Universal Robots PolyScope program: browser.urp

Program browser (installation=cube_dev1 directory=/programs/cube createdIn=5.11.5.1010327 lastSavedIn=5.11.5.1010327 robotSerialNumber=20215500677)
Calibrated DH parameters: a=[0.000204, -0.239222, -0.391845, -0.000001, 0.000022, 0]; d=[0.162722, -355.808559, 353.37206, 2.570385, 0.099741, 0.099629]; alpha=[1.571124, 0.000988, 0.008295, 1.568963, -1.570303, 0]; deltaTheta=[0, -0.973091, 7.204745, 0.05153, 0, 0]
BeforeStart
  MoveJ speed 120 deg/s, acceleration 120 deg/s^2 (useActiveTCP=false) tcp=SandTCP; feature=Point_1
    Waypoint Sand_Base: TCP in base x=-341.949 y=196.192 z=697.874 mm, rx=0 ry=0 rz=-1.5708 rad; joints [-57.163, -82.73, 107.731, 93.373, -53.983, -132.185] deg; TCP offset x=1.003 y=125.541 z=104.154 mm, rx=-0.7854 ry=0 rz=0 rad; feature pose in base x=-341.965 y=196.202 z=697.85 mm, rx=0 ry=0 rz=-1.5843 rad
Robot Program (runOnlyOnce=false)
  Wait Sleep waitTime=0.01
Event  expression=PinsBtn≟ True
  Folder Sand
    MoveL speed 50 mm/s, acceleration 1200 mm/s^2 (useActiveTCP=false) tcp=SandTCP; feature=Base
      MoveDirectionNode (selectedDirection=ZPlus)
        Until TOOL_CONTACT_DETECTION (allowActions=false retraction=0.001 decelerationAcceleration=3 decelerationAngularAcceleration=34.906585)
      URCap Finishing Tool Control (Robotiq_Copilot, Robotiq Inc.) dataModel(ToolOutputNameKey=SanderOn, HackTriggeringContributionIsDefinedMethodKey=true)
    MoveL speed 50 mm/s, acceleration 1200 mm/s^2 (useActiveTCP=true) feature=Base
      Force Simple feature=Base; selection=[0, 0, 1, 0, 0, 0]; wrench=[0, 0, 5, 0, 0, 0]; limitsForce=[0.15, 0.15, 0.15, 1.047198, 1.047198, 1.047198]; limitsMotion=[0.1, 0.1, 0.1, 0.349066, 0.349066, 0.349066]
        MoveDirectionNode (selectedDirection=XMinus)
          Until DISTANCE (allowActions=false deceleration=3 distanceNodeType=BLEND) Distance=0.355; motionParameters(blendRadius=0.025)
        MoveDirectionNode (selectedDirection=YMinus)
          Until DISTANCE (allowActions=false deceleration=3 distanceNodeType=BLEND) Distance=0.335; motionParameters(blendRadius=0.025)
        MoveDirectionNode (selectedDirection=XPlus)
          Until DISTANCE (allowActions=false deceleration=3 distanceNodeType=BLEND) Distance=0.355; motionParameters(blendRadius=0.025)
        MoveDirectionNode (selectedDirection=YPlus)
          Until DISTANCE (allowActions=false deceleration=3 distanceNodeType=STOP) Distance=0.335; motionParameters(blendRadius=0.01)
        URCap Finishing Tool Control (Robotiq_Copilot, Robotiq Inc.) dataModel(FinishingToolStateKey=false, ToolOutputNameKey=SanderOn, HackTriggeringContributionIsDefinedMethodKey=true)
    MoveL speed 90 mm/s, acceleration 1200 mm/s^2 (useActiveTCP=false) tcp=SandTCP; feature=Base
      MoveDirectionNode (selectedDirection=ZMinus)
        Until DISTANCE (allowActions=false deceleration=3 distanceNodeType=BLEND) Distance=0.05; motionParameters(blendRadius=0.003)
  Folder Spray Vert
    MoveJ speed 120 deg/s, acceleration 150 deg/s^2 (useActiveTCP=false) tcp=SprayTCP; feature=Point_1
      Waypoint Spray_Base: TCP in base x=-329.987 y=204.971 z=725 mm, rx=0 ry=0 rz=0.0032 rad; joints [-52.819, -91.06, 108.773, 103.186, -56.031, 43.467] deg; TCP offset x=63.143 y=-107.882 z=84.395 mm, rx=0.6139 ry=0.6139 rz=-1.4822 rad; feature pose in base x=-330 y=205 z=580 mm, rx=0 ry=0 rz=-1.5843 rad
    MoveL speed 90 mm/s, acceleration 1200 mm/s^2 (useActiveTCP=false) tcp=SprayTCP; feature=Base
      MoveDirectionNode (selectedDirection=ZMinus)
        Until DISTANCE (allowActions=false deceleration=3 distanceNodeType=BLEND) Distance=0.075; motionParameters(blendRadius=0.001)
      Set DigitalOutput pin=SprayerOn; digitalValue=1
      MoveDirectionNode (selectedDirection=XMinus)
        Until DISTANCE (allowActions=false deceleration=3 distanceNodeType=BLEND) Distance=0.355; motionParameters(blendRadius=0.001)
      MoveDirectionNode (selectedDirection=YMinus)
        Until DISTANCE (allowActions=false deceleration=3 distanceNodeType=BLEND) Distance=0.33; motionParameters(blendRadius=0.001)
      MoveDirectionNode (selectedDirection=XPlus)
        Until DISTANCE (allowActions=false deceleration=3 distanceNodeType=BLEND) Distance=0.355; motionParameters(blendRadius=0.001)
      MoveDirectionNode (selectedDirection=YPlus)
        Until DISTANCE (allowActions=false deceleration=3 distanceNodeType=BLEND) Distance=0.33; motionParameters(blendRadius=0.001)
      MoveDirectionNode (selectedDirection=XMinus)
        Until DISTANCE (allowActions=false deceleration=3 distanceNodeType=BLEND) Distance=0.05; motionParameters(blendRadius=0.001)
      Set DigitalOutput pin=SprayerOn; digitalValue=0
  MoveJ speed 120 deg/s, acceleration 120 deg/s^2 (useActiveTCP=false) tcp=SandTCP; feature=Point_1
    Waypoint Sand_Base: TCP in base x=-341.949 y=196.192 z=697.874 mm, rx=0 ry=0 rz=-1.5708 rad; joints [-57.163, -82.73, 107.731, 93.373, -53.983, -132.185] deg; TCP offset x=1.003 y=125.541 z=104.154 mm, rx=-0.7854 ry=0 rz=0 rad; feature pose in base x=-341.965 y=196.202 z=697.85 mm, rx=0 ry=0 rz=-1.5843 rad
